// TIA Portal V19 export
FUNCTION_BLOCK "CoilCheckLooseWrap"   // FB21, LAD
TITLE = Detect when coil has loose the wrapping
// Cotrolla quando le spire del rotolo si aprono.
// stored: MemoryReserve 100, SetENOAutomatically false
   VAR_INPUT
      Execute : Bool;
      D_Act : Real;   // Actual coil diameter
      LooseWrap_Delta : Real := 10.0;
      LooseWrap_Time : Time;
   END_VAR
   VAR_OUTPUT
      LooseWrap : Bool;
   END_VAR
   VAR
      On : Bool;
      "M" : Bool;
      D_Min : Real;
      D_Delta : Real;
      TON_Loose { S7_SetPoint := 'True'} : TON_TIME;
   END_VAR
BEGIN

REGION Network 1
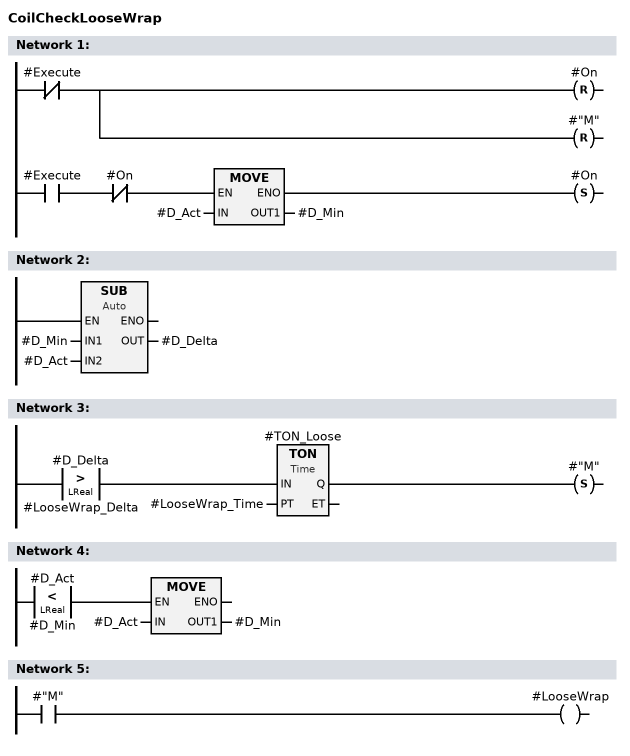
   RUNG wire#powerrail
      I_Contact( #Execute )
      wire#w1
      R_Coil( #On )
   END_RUNG
   RUNG wire#w1
      R_Coil( #"M" )
   END_RUNG
   RUNG wire#powerrail
      Contact( #Execute )
      I_Contact( #On )
      Move(in := #D_Act, out1 => #D_Min)
      S_Coil( #On )
   END_RUNG
   // the same network as SCL:
   IF NOT #Execute THEN
       #On := FALSE;
       #"M" := FALSE;
   END_IF;
   IF #Execute AND NOT #On THEN
       #D_Min := #D_Act;
       #On := TRUE;
   END_IF;
END_REGION

REGION Network 2
   RUNG wire#powerrail
      Sub(in1 := #D_Min, in2 := #D_Act, out => #D_Delta)
   END_RUNG
   // the same network as SCL:
   #D_Delta := #D_Min - #D_Act;
END_REGION

REGION Network 3
   RUNG wire#powerrail
      { S7_Templates := "SrcType := LReal" } GT_Contact(in1 := #D_Delta, in2 := #LooseWrap_Delta)
      { S7_Templates := "time_type := Time" } #TON_Loose.TON(pt := #LooseWrap_Time, et =>)
      S_Coil( #"M" )
   END_RUNG
   // the same network as SCL:
   #TON_Loose(IN := #D_Delta > #LooseWrap_Delta, PT := #LooseWrap_Time);   // TON
   IF #TON_Loose.Q THEN #"M" := TRUE; END_IF;
END_REGION

REGION Network 4
   RUNG wire#powerrail
      { S7_Templates := "SrcType := LReal" } LT_Contact(in1 := #D_Act, in2 := #D_Min)
      Move(in := #D_Act, out1 => #D_Min)
   END_RUNG
   // the same network as SCL:
   IF #D_Act < #D_Min THEN #D_Min := #D_Act; END_IF;
END_REGION

REGION Network 5
   RUNG wire#powerrail
      Contact( #"M" )
      Coil( #LooseWrap )
   END_RUNG
   // the same network as SCL:
   #LooseWrap := #"M";
END_REGION
END_FUNCTION_BLOCK
